// TIA Portal V18 export
TYPE "RCS_CountCycleTime_V1"
   STRUCT
      Count : Struct   // DBX0.0+316*N, N=PM No.-1 / DBX700.0
         OK : Array[0..14] of DInt;
         NG : Array[0..14] of DInt;
         Total : DInt;
         OKHolding : DInt;
         NGHolding : DInt;
         TotalHolding : DInt;
         ClearOK : Bool;
         ClearNG : Bool;
         ClearTotal : Bool;
      END_STRUCT;
      TotalCycleTime : Struct   // DBX138.0+316*N, N=PM No.-1 / DBX850.0
         No : Array[0..21] of Real;
      END_STRUCT;
      MachineCycleTime : Struct   // DBX226.0+316*N, N=PM No.-1 / DBX950.0
         No : Array[0..21] of Real;
      END_STRUCT;
      Num : USInt;
   END_STRUCT;
END_TYPE
